// TIA Portal V20 export
// export: Created 2025-12-01T14:57:05.4056269Z, ExportSetting None, DisplayName Totally Integrated Automation Portal, DisplayVersion V20 Update 3, DisplayName TIA Portal Openness, DisplayVersion V20 Update 3, DisplayName TIA Portal Version Control Interface, DisplayVersion V20 Update 3, DisplayName STEP 7 Professional, DisplayVersion V20 Update 3, DisplayName STEP 7 Safety, DisplayVersion V20 Update 2, DisplayName WinCC Basic/Comfort/Advanced, DisplayVersion V20 Update 3, DisplayName WinCC Professional, DisplayVersion V20 Update 3, DisplayName WinCC Unified, DisplayVersion V20 Update 3
FUNCTION "FC871_NumUTsEnMesa" : Void   // FC871, LAD
{ S7_Optimized_Access := 'FALSE' }
VERSION : 1.0
// stored: AutoNumber false, SetENOAutomatically false
   VAR_INPUT
      Mesa : UInt;
   END_VAR
   VAR_OUTPUT
      NumUTs : UInt;
   END_VAR
   VAR_TEMP
      NumeroUT : UInt;
      AuxNumUTsEnMesa : UInt;
      Relleno : Byte;
      ValorReturn : Int;
   END_VAR
BEGIN

NETWORK
TITLE = ---
////////////////////////////////////////////////////////////////////////////
// --- Reseteo Variable de Salida

      L     0;
      T     #AuxNumUTsEnMesa;  // NumUTs = 0



NETWORK
TITLE = --
////////////////////////////////////////////////////////////////////////////
// --- Comprobacion de que la Mesa tenga UT o No


      L     "DB810_ColasMesas".Colas[#Mesa].UT_PrimeraMesa;
      T     #NumeroUT;

InicioBucleMesa:NOP   0;
      L     #NumeroUT;
      L     0;
      ==I;
      JC    Final;  // No hay UT's ?

      L     1;  // Incrementa el Numero de UTs en la Mesa
      L     #AuxNumUTsEnMesa;
      +I;
      T     #AuxNumUTsEnMesa;

      L     "DB812_UTs_Control".UT[#NumeroUT].UT_SiguienteMesa;
      T     #NumeroUT;

      JU    InicioBucleMesa;



NETWORK
TITLE = ---
// ----------------------------------------------------------------------------
// --- Final de la Funcion

Final:NOP   0;  // Finalizar Funcion
      L     #AuxNumUTsEnMesa;
      T     #NumUTs;


END_FUNCTION
